{attribute 'GeneratedUsingTerminal: EL6201-0000-0017'}
{attribute addProperty BoxType "EL6201-0000-0017"}
{attribute addProperty Id "Slave_29A_DO0BOOL1Slave_29A_DO1BOOL1Slave_29A_DO2BOOL1Slave_29A_DO3BOOL1Slave_29B_DO0BOOL1Slave_29B_DO1BOOL1Slave_29B_DO2BOOL1Slave_29B_DO3BOOL1"}
{attribute addProperty CRC "3427387429"}
{attribute addProperty Size "8"}
TYPE Slave_29_Outputs_CC49C825 :
STRUCT
	{attribute addProperty Name "Slave_29A_DO0"}
	Slave_29A_DO0 : BOOL;
	{attribute addProperty Name "Slave_29A_DO1"}
	Slave_29A_DO1 : BOOL;
	{attribute addProperty Name "Slave_29A_DO2"}
	Slave_29A_DO2 : BOOL;
	{attribute addProperty Name "Slave_29A_DO3"}
	Slave_29A_DO3 : BOOL;
	{attribute addProperty Name "Slave_29B_DO0"}
	Slave_29B_DO0 : BOOL;
	{attribute addProperty Name "Slave_29B_DO1"}
	Slave_29B_DO1 : BOOL;
	{attribute addProperty Name "Slave_29B_DO2"}
	Slave_29B_DO2 : BOOL;
	{attribute addProperty Name "Slave_29B_DO3"}
	Slave_29B_DO3 : BOOL;
END_STRUCT
END_TYPE

(* stored: Version 1.2.0.0, ProductVersion 3.1.4024.9
   DUT Slave_29_Outputs_CC49C825: Id {d279d756-cf4e-4be0-ad86-94ee47f341e3} *)
